(* PLC project Unnamed, Unknown Unnamed 1 *)
(* stored: creationDateTime 2024-11-07T01:46:06, modificationDateTime 2024-11-07T03:23:32 *)

PROGRAM program0
  VAR
    STATE : WORD := 1;
    Traffic_A : WORD := 1;
    Traffic_B : WORD := 2;
    AtoB_Amber : WORD := 4;
    BtoA_Amber : WORD := 8;
    A_Crossing_A_Amber : WORD := 16;
    A_Crossing_A : WORD := 32;
    A_Crossing_B_Amber : WORD := 64;
    A_Crossing_B : WORD := 128;
    B_Crossing_A_Amber : WORD := 256;
    B_Crossing_A : WORD := 512;
    B_Crossing_B_Amber : WORD := 1024;
    B_Crossing_B : WORD := 2048;
    A_Crossing_Latch : BOOL := false;
    B_Crossing_Latch : BOOL := false;
  END_VAR
  VAR
    Change_Button AT %IX0.5 : BOOL;
    Cross_A_Button AT %IX0.6 : BOOL;
    Cross_B_Button AT %IX0.7 : BOOL;
    Green_A_LED AT %QX0.0 : BOOL;
    Amber_A_LED AT %QX0.1 : BOOL;
    Red_A_LED AT %QX0.2 : BOOL;
    Green_B_LED AT %QX0.3 : BOOL;
    Amber_B_LED AT %QX0.4 : BOOL;
    Red_B_LED AT %QX0.5 : BOOL;
    Cross_A_LED AT %QX0.6 : BOOL;
    Cross_B_LED AT %QX0.7 : BOOL;
  END_VAR
  VAR
    Amber_Dwell : TIME := T#2s;
    Traffic_Dwell : TIME := T#5s;
    Crossing_Dwell : TIME := T#3s;
    TON0 : TON;
    TON1 : TON;
    TON2 : TON;
    TON3 : TON;
    TON4 : TON;
    TON5 : TON;
    TON6 : TON;
    TON7 : TON;
    TON8 : TON;
    TON9 : TON;
    TON10 : TON;
    TON11 : TON;
    TON12 : TON;
  END_VAR
  VAR  (* added by the conversion: wires and edge detectors of the diagram *)
    _EQ23_OUT : BOOL;
    _EQ20_OUT : BOOL;
    _EQ75_OUT : BOOL;
    _EQ91_OUT : BOOL;
    _EQ107_OUT : BOOL;
    _EQ123_OUT : BOOL;
  END_VAR

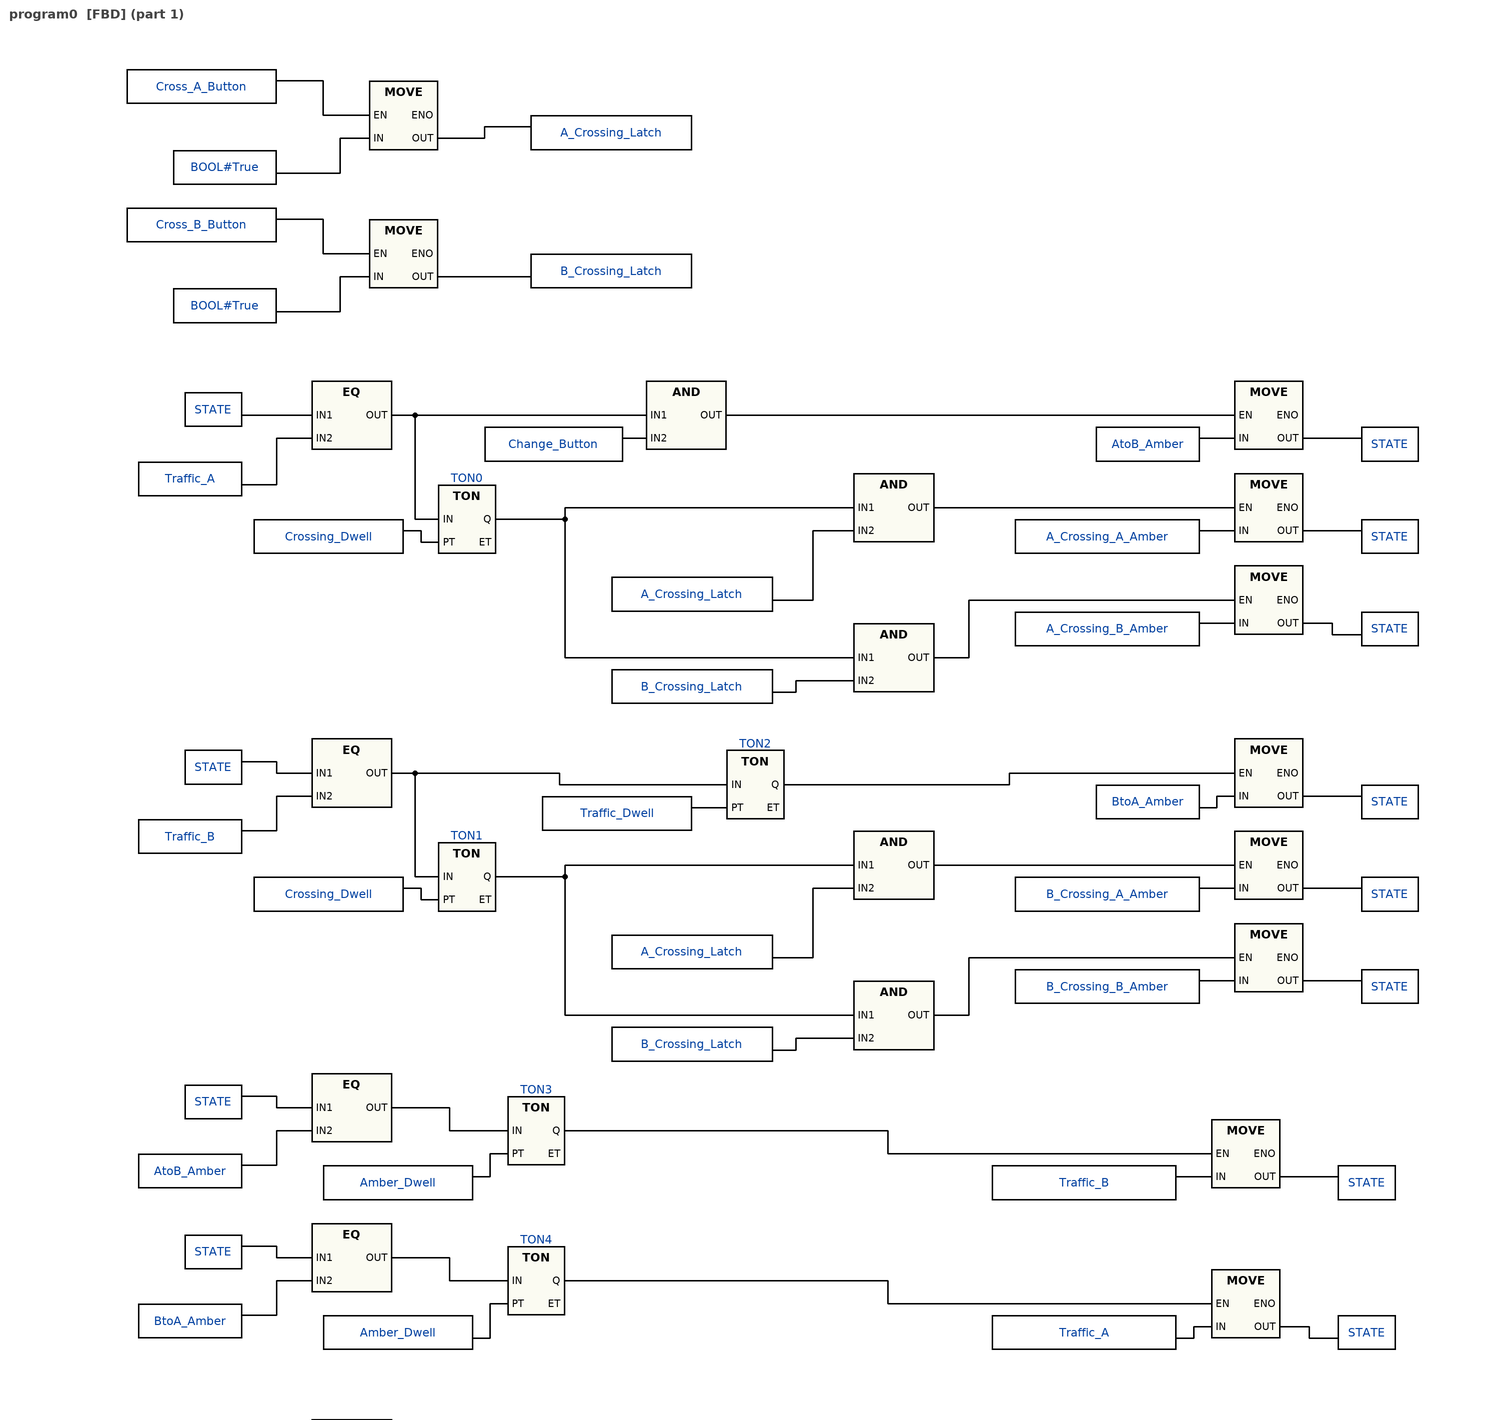
(* FBD diagram, written out as Structured Text *)
IF Cross_A_Button THEN A_Crossing_Latch := BOOL#True; END_IF;
IF Cross_B_Button THEN B_Crossing_Latch := BOOL#True; END_IF;
_EQ23_OUT := STATE = Traffic_A;
IF _EQ23_OUT AND Change_Button THEN STATE := AtoB_Amber; END_IF;
TON0(IN := _EQ23_OUT, PT := Crossing_Dwell);
IF TON0.Q AND A_Crossing_Latch THEN STATE := A_Crossing_A_Amber; END_IF;
IF TON0.Q AND B_Crossing_Latch THEN STATE := A_Crossing_B_Amber; END_IF;
_EQ20_OUT := STATE = Traffic_B;
TON2(IN := _EQ20_OUT, PT := Traffic_Dwell);
IF TON2.Q THEN STATE := BtoA_Amber; END_IF;
TON1(IN := _EQ20_OUT, PT := Crossing_Dwell);
IF TON1.Q AND A_Crossing_Latch THEN STATE := B_Crossing_A_Amber; END_IF;
IF TON1.Q AND B_Crossing_Latch THEN STATE := B_Crossing_B_Amber; END_IF;
TON3(IN := STATE = AtoB_Amber, PT := Amber_Dwell);
IF TON3.Q THEN STATE := Traffic_B; END_IF;
TON4(IN := STATE = BtoA_Amber, PT := Amber_Dwell);
IF TON4.Q THEN STATE := Traffic_A; END_IF;
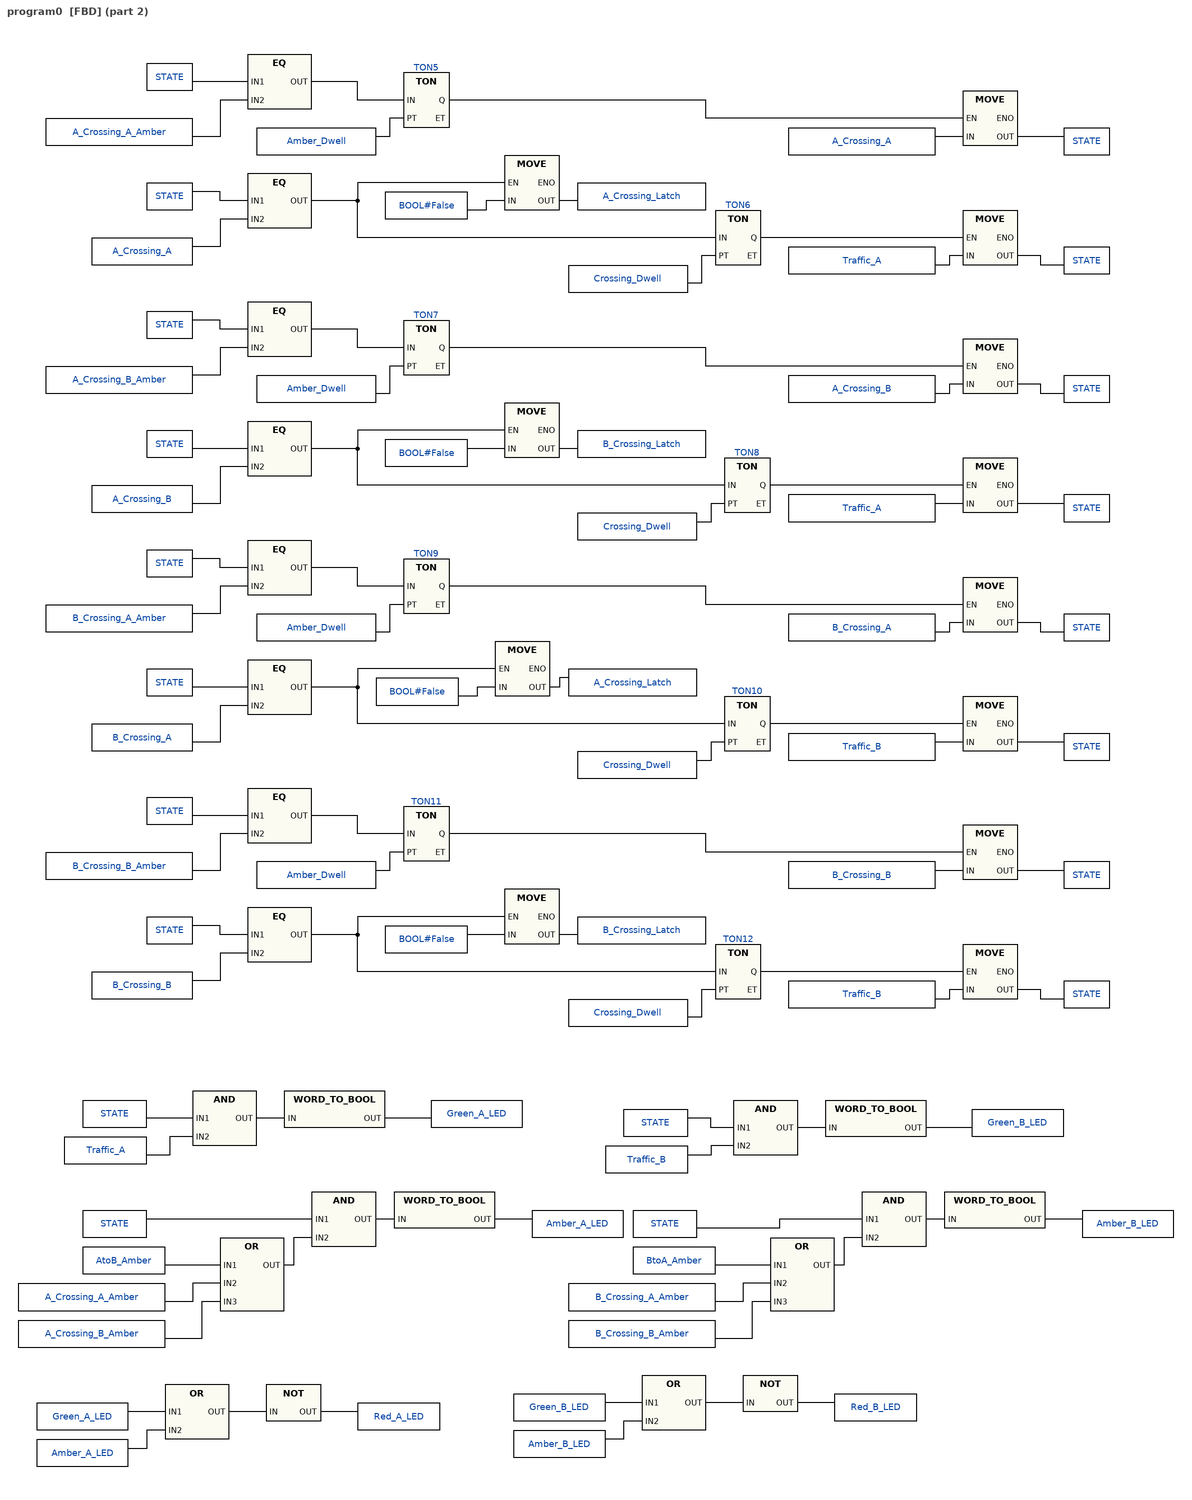
TON5(IN := STATE = A_Crossing_A_Amber, PT := Amber_Dwell);
IF TON5.Q THEN STATE := A_Crossing_A; END_IF;
_EQ75_OUT := STATE = A_Crossing_A;
TON6(IN := _EQ75_OUT, PT := Crossing_Dwell);
IF TON6.Q THEN STATE := Traffic_A; END_IF;
TON7(IN := STATE = A_Crossing_B_Amber, PT := Amber_Dwell);
IF TON7.Q THEN STATE := A_Crossing_B; END_IF;
_EQ91_OUT := STATE = A_Crossing_B;
TON8(IN := _EQ91_OUT, PT := Crossing_Dwell);
IF TON8.Q THEN STATE := Traffic_A; END_IF;
TON9(IN := STATE = B_Crossing_A_Amber, PT := Amber_Dwell);
IF TON9.Q THEN STATE := B_Crossing_A; END_IF;
_EQ107_OUT := STATE = B_Crossing_A;
TON10(IN := _EQ107_OUT, PT := Crossing_Dwell);
IF TON10.Q THEN STATE := Traffic_B; END_IF;
TON11(IN := STATE = B_Crossing_B_Amber, PT := Amber_Dwell);
IF TON11.Q THEN STATE := B_Crossing_B; END_IF;
_EQ123_OUT := STATE = B_Crossing_B;
TON12(IN := _EQ123_OUT, PT := Crossing_Dwell);
IF TON12.Q THEN STATE := Traffic_B; END_IF;
IF _EQ75_OUT THEN A_Crossing_Latch := BOOL#False; END_IF;
IF _EQ107_OUT THEN A_Crossing_Latch := BOOL#False; END_IF;
IF _EQ91_OUT THEN B_Crossing_Latch := BOOL#False; END_IF;
IF _EQ123_OUT THEN B_Crossing_Latch := BOOL#False; END_IF;
Green_A_LED := WORD_TO_BOOL(STATE AND Traffic_A);
Green_B_LED := WORD_TO_BOOL(STATE AND Traffic_B);
Amber_A_LED := WORD_TO_BOOL(STATE AND (AtoB_Amber OR A_Crossing_A_Amber OR A_Crossing_B_Amber));
Amber_B_LED := WORD_TO_BOOL(STATE AND (BtoA_Amber OR B_Crossing_A_Amber OR B_Crossing_B_Amber));
Red_A_LED := NOT (Green_A_LED OR Amber_A_LED);
Red_B_LED := NOT (Green_B_LED OR Amber_B_LED);
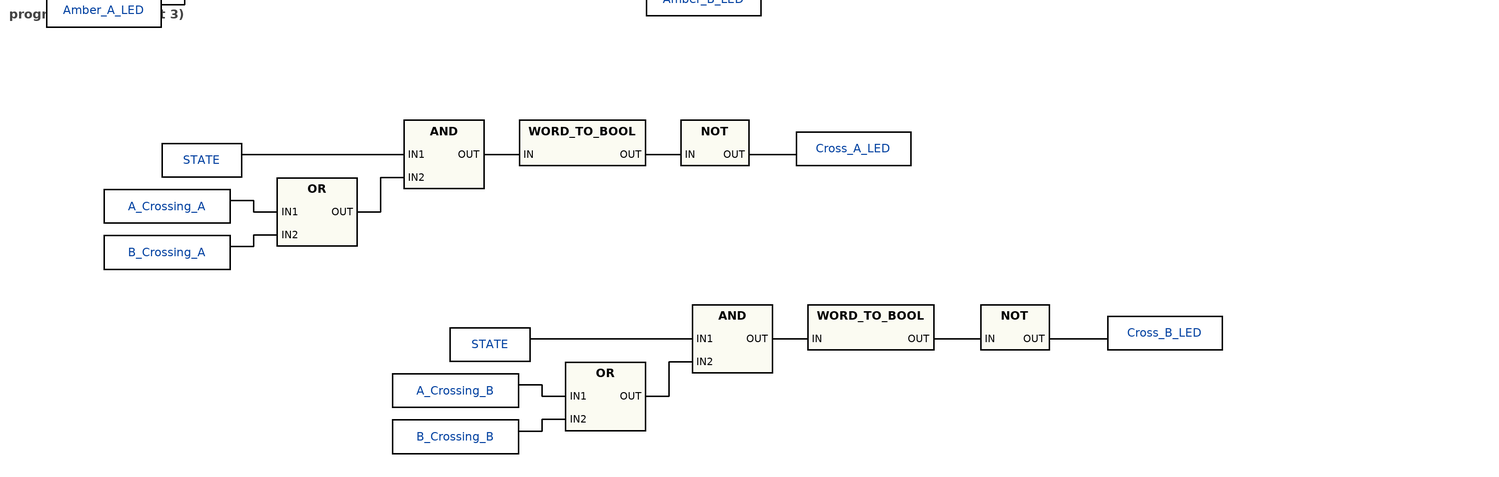
Cross_A_LED := NOT WORD_TO_BOOL(STATE AND (A_Crossing_A OR B_Crossing_A));
Cross_B_LED := NOT WORD_TO_BOOL(STATE AND (A_Crossing_B OR B_Crossing_B));
END_PROGRAM

CONFIGURATION Config0
  RESOURCE Res0 ON PLC
    TASK task0(INTERVAL := T#20ms, PRIORITY := 0);
    PROGRAM instance0 WITH task0 : program0;
  END_RESOURCE
END_CONFIGURATION
